FUNCTION_BLOCK FB_EventLogger
VAR
 	EventBuffer : ARRAY [1..MAXIMUM_SIZE_OF_EVENT_BUFFER] OF St_Event ;
	CurrentEventBufferIndex : INT := 0 ;
	
	_PersistentEventStorage : I_PersistentEventStorage ;
END_VAR

VAR CONSTANT
	MAXIMUM_SIZE_OF_EVENT_BUFFER : INT := 100 ;
END_VAR



_PersistentEventStorage.StoreEvent(stEvent :=  EventBuffer[CurrentEventBufferIndex]) ;

METHOD PUBLIC AddEvent : BOOL
VAR_INPUT
	eEventType : E_EventType ;
	eEventSeverity : TcEventSeverity ;
	nEventIdentiy : UDINT ;
	sEventText : STRING (255) ;
END_VAR
IF NOT IsEventBufferFull () THEN
	CurrentEventBufferIndex := CurrentEventBufferIndex +1 ;
	EventBuffer[CurrentEventBufferIndex].eEventType 	:= eEventType 		;
	EventBuffer[CurrentEventBufferIndex].eEventSeverity := eEventSeverity 	;
	EventBuffer[CurrentEventBufferIndex].nEventIdentiy 	:= nEventIdentiy	;
	EventBuffer[CurrentEventBufferIndex].sEventText 	:= sEventText		;
	F_UpdateEventTimeStampWithSystemTime(stEvent := EventBuffer[CurrentEventBufferIndex]);
		
	AddEvent := TRUE ;	
ELSE
	AddEvent := FALSE ;
END_IF

_PersistentEventStorage.StoreEvent(stEvent := EventBuffer[CurrentEventBufferIndex]) ;
END_METHOD

METHOD FB_init : BOOL
VAR_INPUT
	bInitRetains : BOOL; // if TRUE, the retain variables are initialized (warm start / cold start)
	bInCopyCode : BOOL;  // if TRUE, the instance afterwards gets moved into the copy code (online change)
	
	iPersistentEventStorage : I_PersistentEventStorage ;
END_VAR

_PersistentEventStorage := iPersistentEventStorage ;
END_METHOD

METHOD PRIVATE IsEventBufferFull : BOOL
VAR_INPUT
	
END_VAR
IF (CurrentEventBufferIndex + 1) > MAXIMUM_SIZE_OF_EVENT_BUFFER THEN
	IsEventBufferFull := TRUE ;
ELSE
	IsEventBufferFull := FALSE ;
END_IF
END_METHOD

END_FUNCTION_BLOCK

(* stored: Version 1.1.0.1, ProductVersion 3.1.4024.12
   POU FB_EventLogger: Id {fa4b927c-8474-469a-8f63-9bb4167680e3}, SpecialFunc None
   Method AddEvent: Id {d4535e1b-00c3-4a75-bac1-b7fa877c881e}
   Method FB_init: Id {d76d3788-a0f3-4cd6-9353-6321b0b9e1a5}
   Method IsEventBufferFull: Id {638c9b8a-aa80-4658-8c0d-5bd2bc252597} *)
